FUNCTION_BLOCK IN_ANY (* Data input from TextField *)
  (* Standard: 61499-1; Classification: GUI *)
  (* Version 0.1, 2002-05-03, JHC, Rockwell Automation, Made QI initial value = true. *)
  (* Version 0.0, 2001-05-31, JHC, Rockwell Automation *)
  (* Compiler header: package fb.rt.hmi; import java.awt.*; *)
  (* Compiler Java IBM VisualAge 3.0 *)
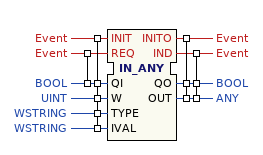
  EVENT_INPUT
    INIT WITH QI, W, TYPE, IVAL;
    REQ WITH QI;
  END_EVENT
  EVENT_OUTPUT
    INITO WITH QO, OUT;
    IND WITH QO, OUT;
  END_EVENT
  VAR_INPUT
    QI : BOOL := true;
    W : UINT := 10; (* TextField width in chars *)
    TYPE : WSTRING := "ANY"; (* Data type name *)
    IVAL : WSTRING;
  END_VAR
  VAR_OUTPUT
    QO : BOOL; (* 1=OK,0=Error *)
    OUT : ANY;
  END_VAR
  SERVICE IN_ANY/TextField
    SEQUENCE normal_initialization
      IN_ANY.INIT+(IVAL) -> TextField.initialize(IVAL) -> OUT.initialize(IVAL) -> IN_ANY.INITO+(OUT);
    END_SEQUENCE
    SEQUENCE initialization_inhibited
      IN_ANY.INIT-() -> IN_ANY.INITO-();
    END_SEQUENCE
    SEQUENCE data_request
      IN_ANY.REQ+() -> TextField.getText() -> OUT.initialize(text) -> IN_ANY.IND+(OUT);
    END_SEQUENCE
    SEQUENCE data_request_error
      IN_ANY.REQ+() -> TextField.getText() -> TextField.setText(errorMessage);
    END_SEQUENCE
    SEQUENCE data_request_inhibited
      IN_ANY.REQ-() -> IN_ANY.IND-();
    END_SEQUENCE
    SEQUENCE user_data_entered
      TextField.dataEntered() -> OUT.initialize(text) -> IN_ANY.IND+(OUT);
    END_SEQUENCE
    SEQUENCE user_data_error
      TextField.dataEntered() -> TextField.setText(errorMessage);
    END_SEQUENCE
  END_SERVICE
END_FUNCTION_BLOCK
